# EPICS substitutions: iocBoot/ioc4idHHLM/substitutions/canberra_13.substitutions
file "$(MCA)/mcaApp/Db/simple_mca.db"
{
pattern
{P           M       DTYP           INP         PREC  CHANS}
{4idHHLM:med:   mca1  "asynMCA"   "@asyn(AIM2/1 0)"    3  2048}
{4idHHLM:med:   mca2  "asynMCA"   "@asyn(AIM2/1 1)"    3  2048}
{4idHHLM:med:   mca3  "asynMCA"   "@asyn(AIM2/1 2)"    3  2048}
{4idHHLM:med:   mca4  "asynMCA"   "@asyn(AIM2/2 0)"    3  2048}
{4idHHLM:med:   mca5  "asynMCA"   "@asyn(AIM2/2 1)"    3  2048}
{4idHHLM:med:   mca6  "asynMCA"   "@asyn(AIM2/2 2)"    3  2048}
{4idHHLM:med:   mca7  "asynMCA"   "@asyn(AIM3/1 0)"    3  2048}
{4idHHLM:med:   mca8  "asynMCA"   "@asyn(AIM3/1 1)"    3  2048}
{4idHHLM:med:   mca9  "asynMCA"   "@asyn(AIM3/1 2)"    3  2048}
{4idHHLM:med:   mca10 "asynMCA"   "@asyn(AIM3/2 0)"    3  2048}
{4idHHLM:med:   mca11 "asynMCA"   "@asyn(AIM3/3 1)"    3  2048}
{4idHHLM:med:   mca12 "asynMCA"   "@asyn(AIM3/4 2)"    3  2048}
{4idHHLM:med:   mca13 "asynMCA"   "@asyn(AIM3/2 3)"    3  2048}
{4idHHLM:med:   mca0  "Soft Channel"   ""     3  2048}
}

file "$(MCA)/mcaApp/Db/icb_amp.db"
{
pattern
{P			AMP		PORT}
{4idHHLM:med:	amp1	"icbAmp1"}
{4idHHLM:med:	amp2	"icbAmp2"}
{4idHHLM:med:	amp3	"icbAmp3"}
{4idHHLM:med:	amp4	"icbAmp4"}
{4idHHLM:med:	amp5	"icbAmp5"}
{4idHHLM:med:	amp6	"icbAmp6"}
{4idHHLM:med:	amp7	"icbAmp7"}
{4idHHLM:med:	amp8	"icbAmp8"}
{4idHHLM:med:	amp9	"icbAmp9"}
{4idHHLM:med:	amp10	"icbAmp10"}
{4idHHLM:med:	amp11	"icbAmp11"}
{4idHHLM:med:	amp12	"icbAmp12"}
{4idHHLM:med:	amp13	"icbAmp13"}
}

file "$(MCA)/mcaApp/Db/icb_adc.db"
{
pattern
{P			ADC		PORT}
{4idHHLM:med:	adc1	"icbAdc1"}
{4idHHLM:med:	adc2	"icbAdc2"}
{4idHHLM:med:	adc3	"icbAdc3"}
{4idHHLM:med:	adc4	"icbAdc4"}
}

file "$(MCA)/mcaApp/Db/icb_hvps.db"
{
pattern
{P			HVPS	LIMIT	PORT}
{4idHHLM:med:	hvps1	1000	"icbHvps1"}
}
